FUNCTION_BLOCK CSV_WRITER_9 (* Service Interface Function Block Type *)
  (* Description: Copyright (c) 2012 ACIN This program and the accompanying materials are made available under the terms of the Eclipse Public License 2.0 which is available at https://www.eclipse.org/legal/epl-2.0/ SPDX-License-Identifier: EPL-2.0 *)
  (* Version 1.0, 2012-06-16, Alois Zoitl, ACIN *)
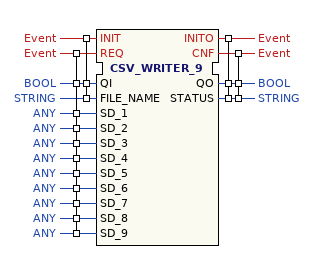
  EVENT_INPUT
    INIT WITH QI, FILE_NAME; (* Service Initialization *)
    REQ WITH QI, SD_1, SD_2, SD_3, SD_4, SD_5, SD_6, SD_7, SD_8, SD_9; (* Service Request *)
  END_EVENT
  EVENT_OUTPUT
    INITO WITH QO, STATUS; (* Initialization Confirm *)
    CNF WITH QO, STATUS; (* Confirmation of Requested Service *)
  END_EVENT
  VAR_INPUT
    QI : BOOL; (* Event Input Qualifier *)
    FILE_NAME : STRING; (* Service Parameters *)
    SD_1 : ANY; (* Output data to resource *)
    SD_2 : ANY;
    SD_3 : ANY;
    SD_4 : ANY;
    SD_5 : ANY;
    SD_6 : ANY;
    SD_7 : ANY;
    SD_8 : ANY;
    SD_9 : ANY;
  END_VAR
  VAR_OUTPUT
    QO : BOOL; (* Event Output Qualifier *)
    STATUS : STRING; (* File access status *)
  END_VAR
  SERVICE APPLICATION/RESOURCE (* Service Interface Function Block Type *)
    SEQUENCE normal_establishment
      APPLICATION.INIT+(FILE_NAME) -> APPLICATION.INITO+(STATUS);
    END_SEQUENCE
    SEQUENCE unsuccessful_establishment
      APPLICATION.INIT+(FILE_NAME) -> APPLICATION.INITO-(STATUS);
    END_SEQUENCE
    SEQUENCE request_confirm
      APPLICATION.REQ+(SD_1,SD_2,SD_3,SD_4,SD_5,SD_6,SD_7,SD_8,SD_9) -> APPLICATION.CNF+(STATUS);
    END_SEQUENCE
    SEQUENCE request_inhibited
      APPLICATION.REQ-(SD_1,SD_2,SD_3,SD_4,SD_5,SD_6,SD_7,SD_8,SD_9) -> APPLICATION.CNF-(STATUS);
    END_SEQUENCE
    SEQUENCE request_error
      APPLICATION.REQ+(SD_1,SD_2,SD_3,SD_4,SD_5,SD_6,SD_7,SD_8,SD_9) -> APPLICATION.CNF-(STATUS);
    END_SEQUENCE
    SEQUENCE application_initiated_termination
      APPLICATION.INIT-() -> APPLICATION.INITO-(STATUS);
    END_SEQUENCE
  END_SERVICE
END_FUNCTION_BLOCK
